INTERFACE ITF_Control1_HMI_Connector_View EXTENDS ITF_BaseControlElement_HMI_Connector_View

END_INTERFACE

(* stored: Version 1.1.0.1
   Itf ITF_Control1_HMI_Connector_View: Id {7a822abb-28d6-024c-0363-ce2b6d11dc02} *)
